        !Trava Produto
        SetDO \Sync, DO_Rc_Fixação_Peça, 0;
        SetDO \Sync, DO_Av_Fixação_Peça, 1;
        !Wait sensores avançado
        WaitTime 1;
        WaitDI DI_Fixa_Peça_1_Rc, 0\MaxTime:= 5\TimeFlag:=timeout_av1;
        WaitDI DI_Fixa_Peça_2_Rc, 0\MaxTime:= 5\TimeFlag:=timeout_av2;
        WaitDI DI_Fixa_Peça_1_Av, 1\MaxTime:= 5\TimeFlag:=timeout_av3;
        WaitDI DI_Fixa_Peça_2_Av, 1\MaxTime:= 5\TimeFlag:=timeout_av4;
        IF (timeout_av1 OR timeout_av2 OR timeout_av3 OR timeout_av4) = TRUE THEN
            PulseDO\PLength:=1, PN_OUT_DO_Cil_NAv;
            TPWrite "Supervisao Sensores, Travas não Avançaram";
            Stop;
            GOTO init_tp;
        ENDIF

    ENDPROC

    !*************************************************************************************************************************
    !Rotinas de Garra: Destravar (Recuar Index Cilindros)
    !*************************************************************************************************************************
    PROC GARRA_DestravarProduto()
    init_dp:
        SetDO PN_OUT_DO_Cil_NRc, 0;

        !Destrava produto na garra
        SetDO \Sync, DO_Av_Fixação_Peça, 0;
        SetDO \Sync, DO_Rc_Fixação_Peça, 1;
        WaitDI DI_Fixa_Peça_1_Av, 0\MaxTime:= 5\TimeFlag:=timeout_rc1;
        WaitDI DI_Fixa_Peça_2_Av, 0\MaxTime:= 5\TimeFlag:=timeout_rc2;
        WaitDI DI_Fixa_Peça_1_Rc, 1\MaxTime:= 5\TimeFlag:=timeout_rc3;
        WaitDI DI_Fixa_Peça_2_Rc, 1\MaxTime:= 5\TimeFlag:=timeout_rc4;
        IF (timeout_rc1 OR timeout_rc2 OR timeout_rc3 OR timeout_rc4) = TRUE THEN
            PulseDO\PLength:=1, PN_OUT_DO_Cil_NRc;
            TPWrite "Supervisao Sensores, Travas não Recuaram";
            Stop;
            GOTO init_dp;
        ENDIF
    ENDPROC

    !*************************************************************************************************************************
    !Rotinas de Garra: Validar Sensor Laser
    !*************************************************************************************************************************
    PROC GARRA_VerificarLaser()
     inicio:
        IF DInput (DI_Pres_Peça_Berço_1) = 0 AND DInput (DI_Pres_Peça_Berço_2) = 1 GOTO Fim;

        PulseDO\PLength:=1, PN_OUT_Produto_Existente;
        TPErase;
        TPWrite "Sensor de presença de peça no berço acionado. Verifique";
        Stop;
        GOTO inicio;

    Fim:
        SetDO PN_OUT_Produto_Existente, 0;
    ENDPROC

    !*************************************************************************************************************************
    !Rotinas de Garra: Validar sensores garra / Garantir que a garra está vazia
    !*************************************************************************************************************************
    PROC GARRA_VerificarGarraVazia()
    !Verifica se robô tem peça na garra ou não

    Verifica:
        IF DI_Pres_Peça_Garra_2 = 1 AND DI_Pres_Peça_Garra_1 = 0 THEN
            GOTO Fim;
        ELSE
            TPErase;
            TPWrite "Deposite manualmente o produto encontrado na garra e reinicie o ciclo";
            TPWrite "Após depositar o produto, adicionar código do produto na IHM";
            IF GInput (PN_IN_Numero_Programa) = 2 THEN
                TPWrite "Programa 'Pega na Esteira de Entrada' necessita de garra vazia para iniciar";
                PulseDO\PLength:=2, PN_OUT_Pos_Home_Manual;
            ELSEIF GInput (PN_IN_Numero_Programa) = 4 THEN
                TPWrite "Programa 'Pega Peça no Buffer' necessita de garra vazia para iniciar";
                PulseDO\PLength:=2, PN_OUT_Pos_Home_Manual;
            ENDIF
            WaitUntil DI_Pres_Peça_Garra_2 = 1 AND DI_Pres_Peça_Garra_1 = 0;
            GOTO Verifica;
        ENDIF
    Fim:
    ENDPROC


    !*************************************************************************************************************************
    !Rotinas de Garra: Define Grip Load da família
    !*************************************************************************************************************************
    PROC GARRA_ConfigurarCarga(Num f)
        TEST f
			CASE 1:
				GripLoad lFamilia_1;
			CASE 2:
				GripLoad lFamilia_2;
			CASE 3:
				GripLoad lFamilia_3;
			CASE 4:
				GripLoad lFamilia_4;

			DEFAULT:
				!Erro
				MsgBoxStop("Número da Família recebida pelo CLP Inexistente!");
				EXIT;
		ENDTEST
    ENDPROC

    !*************************************************************************************************************************
    !Função para ser chamada pela manutenção (retorno para home)
    !*************************************************************************************************************************
    PROC EXTRAS_PosicionaHomeManual()
        VAR robtarget pPosição_Atual;
        VAR num nAux_Limite_Low;

        !Movimente manualmente o robô até uma posição em que esteja livre de colisão e acione os comandos abaixo.

    verif:
        pPosição_Atual := CRobT(\Tool:=tGarra \WObj:=wobj0);

        nAux_Limite_Low := 550;
        IF (pPosição_Atual.trans.z > nAux_Limite_Low) THEN
            GOTO DoHome;
        ELSE
            TPErase;
            TPWrite "Posicione Robô mais Alto";
            Stop\NoRegain;
            GOTO verif;
        ENDIF

    DoHome:
        MoveJ pPosicaoHome, sMov_Geral_Sem_Produto, fine, tGarra \WObj:=wobj0;
        SetDO PN_OUT_Pos_Home_Manual, 0;


    ENDPROC

!*****************************************************************************************************************************
    !FUNÇÕES EXTRAS: Teste de Posições no Buffer (Área "A" - à esquerda do robô quando de costas para as esteiras )
    !*****************************************************************************************************************************
    PROC EXTRAS_TesteBufferAreas()
        !Este programa irá enviar o robô à partir de home, index-por-index (de trás para frente) relacionados às áreas do Buffer


        VAR num f;
        VAR num zLoopValida;
        VAR num zFinal;
        VAR num i_ini;
        VAR num InputUsuarioArea;
        VAR num InputUsuario3Opcoes;

        VAR bool InputUsuarioSim;
        VAR bool InputUsuarioDescer;
        VAR bool init;
        VAR bool SaiLoopValida;
        VAR bool InputUsuarioCrescente;

        VAR robtarget RT_PosicaoBuffer;
        VAR robtarget RT_PosicaoAuxiliar;
        VAR jointtarget RJ_PosicaoAuxiliar;

        VAR speeddata SPEEDDATA_VelocidadeAuxiliar;
        VAR string STR_AreaSelecionada;

        !Considerações iniciais
        TPErase;
        TPWrite "Este programa irá enviar o robô index-por-index. Já deve existir peça na garra!";
        TPWrite "Para sobrescrever os pontos, garanta que foram renomeados de CONST para PERS.";
        Stop;
        TPErase;

        StartMove;

        !Pergunta ao usuário qual família
        f := MsgBoxInputUsuarioModelo();

        !Se usuário cancelou, encerra
        IF f = 5 THEN
            EXIT;
        ENDIF

        !Pergunta ao usuário qual área de trabalho
        !(1=Pallet Entrada, 2=Pallet Saída, 3=A, 4=B, 5=C)
        InputUsuarioArea := MsgBoxInputUsuarioWorkObject();

        TEST InputUsuarioArea
            CASE 3:
                STR_AreaSelecionada := "A";
            CASE 4:
                STR_AreaSelecionada := "B";
            CASE 5:
                STR_AreaSelecionada := "C";
            DEFAULT:
                MsgBoxStop("Função Ainda Não Suportada!");
                EXIT;
        ENDTEST

        !Pergunta ao usuário por qual index começar
        gNUM_IteradorBuffer := MsgBoxInputNumericoUsuario("Qual local do Buffer iniciar? (de 1 a 99). 0 = 'Cancelar'");

        !Se usuário cancelou, encerra
        IF (gNUM_IteradorBuffer = 0) OR (gNUM_IteradorBuffer > 99) THEN
            EXIT;
        ENDIF

        !Pergunta ao usuário se adiciona ou decrementa os indexes
        InputUsuarioCrescente := MsgBoxSimNao("Iterar de forma Crescente ou Decrescente?", "Crescente", "Decrescente");

        !Inicializa Parametros
        AccSet 60, 40;
        MotionSup \On \TuneValue:= 200;

        !Vai pra Home?
        IF MsgBoxSimNao("Retornar para Home?", "Sim", "Não") THEN
            SPEEDDATA_VelocidadeAuxiliar := GetSpeedDataFamilia("SPEEDDATA_Geral", f);
            MoveJ pPosicaoHome, SPEEDDATA_VelocidadeAuxiliar, z500, tGarra\WObj:=wobj0;
        ENDIF

        init := TRUE;

        !index-por-index (de trás para frente)
        WHILE gNUM_IteradorBuffer > 0 DO
            !Verifica se index corresponde à área selecionada (A, B ou C)
            IF GetAreaBuffer(gNUM_IteradorBuffer) <> STR_AreaSelecionada THEN
                GOTO break_a;
            ENDIF

            !Se família HL8, verifica se posição corresponde
            IF (f = 4) AND (NOT IsIndexHL8(gNUM_IteradorBuffer)) THEN
                GOTO break_a;
            ENDIF


            !Lê o valor da posição através da descrição da tag
            RT_PosicaoBuffer := GetPosicaoBuffer(gNUM_IteradorBuffer, f);

            !Lê qual o frame da posição atual
            gWOBJDATA_FrameAtual := GetWObjBuffer(gNUM_IteradorBuffer);


            IF init THEN
                !Vai para centro de massa
                !Ponto intermediario centro de massa
                RT_PosicaoAuxiliar := RT_PosicaoBuffer;
        	    RJ_PosicaoAuxiliar := CalcJointT(RT_PosicaoAuxiliar, tGarra \WObj:=gWOBJDATA_FrameAtual);
                RJ_PosicaoAuxiliar.robax.rax_2 := jposRecolhidoEsteira.robax.rax_2;
                RJ_PosicaoAuxiliar.robax.rax_3 := jposRecolhidoEsteira.robax.rax_3;
                RJ_PosicaoAuxiliar.robax.rax_4 := jposRecolhidoEsteira.robax.rax_4;
                RJ_PosicaoAuxiliar.robax.rax_5 := jposRecolhidoEsteira.robax.rax_5;

                SPEEDDATA_VelocidadeAuxiliar := GetSpeedDataFamilia("SPEEDDATA_Geral", f);
                MoveAbsJ RJ_PosicaoAuxiliar, SPEEDDATA_VelocidadeAuxiliar, z500, tGarra\WObj:=gWOBJDATA_FrameAtual;
                init := false;
            ENDIF


            !Vai para posição acima do local de deposita
            RT_PosicaoAuxiliar := RT_PosicaoBuffer;
            RT_PosicaoAuxiliar.trans.z := RT_PosicaoAuxiliar.trans.z + 450;

            SPEEDDATA_VelocidadeAuxiliar := GetSpeedDataFamilia("SPEEDDATA_Geral", f);
            MoveL RT_PosicaoAuxiliar, SPEEDDATA_VelocidadeAuxiliar, z20, tGarra\WObj:=gWOBJDATA_FrameAtual;

            !Ponto acima do berço (seguro)
            RT_PosicaoAuxiliar := RT_PosicaoBuffer;
            RT_PosicaoAuxiliar.trans.z := RT_PosicaoAuxiliar.trans.z + 300;

            SPEEDDATA_VelocidadeAuxiliar := GetSpeedDataFamilia("SPEEDDATA_Geral", f);
            MoveL RT_PosicaoAuxiliar, SPEEDDATA_VelocidadeAuxiliar, z50, tGarra\WObj:=gWOBJDATA_FrameAtual;

            !Aqui já temos uma boa idéia se irá entrar sem bater.
            !Se precisar de algum ajuste, usuário poderá fazê-lo e confirmar
            StopMove;

            ClearPath;
            !InputUsuarioSim := MsgBoxSimNao("Ajustar a posição de entrada e confirmar para prosseguir", "Prosseguir", "Cancelar");
            MsgBoxStop("Ajustar a posição de entrada. Aperte 'Play' para prosseguir");
            StartMove;

            !Ponto de aproximação
            AccSet 30, 40;
            MotionSup \On \TuneValue:= 80;

            !Parte-se do princípio que usuário alterou a posição relativa
            !Pega posição atual e altera Z para bater com a posição do buffer
            RT_PosicaoAuxiliar := CRobT(\Tool:=tGarra \WObj:=gWOBJDATA_FrameAtual);
            RT_PosicaoAuxiliar.trans.z := RT_PosicaoBuffer.trans.z + 55;

            SPEEDDATA_VelocidadeAuxiliar := GetSpeedDataFamilia("SPEEDDATA_AtaqueLinSeg", f);
            MoveL RT_PosicaoAuxiliar, SPEEDDATA_VelocidadeAuxiliar, z0, tGarra\WObj:=gWOBJDATA_FrameAtual;

            !Registra Z original do ponto em questão
            zFinal := RT_PosicaoBuffer.trans.z;

            !Aqui já temos uma boa idéia se irá entrar sem bater.
            !Se precisar de algum ajuste, usuário poderá fazê-lo e confirmar

            StopMove;
            ClearPath;
            InputUsuario3Opcoes := MsgBox3Opcoes("Ajustar posição. Selecionar Opção:", "Descer 5mm", "Pular", "Descer Posição Final");
            StartMove;

            If InputUsuario3Opcoes <> 2 THEN
                SaiLoopValida := FALSE;
            ELSE
                SaiLoopValida := TRUE;
            ENDIF

            !Agora entra em loop, decrementando Z e perguntando input do usuário
            WHILE NOT SaiLoopValida DO

                !Parte-se do princípio que usuário alterou a posição relativa
                !Pega posição atual e altera Z para bater com a posição do buffer
                RT_PosicaoAuxiliar := CRobT(\Tool:=tGarra \WObj:=gWOBJDATA_FrameAtual);

                TEST InputUsuario3Opcoes
                    CASE 1: !Desce 5mm
                        RT_PosicaoAuxiliar.trans.z := RT_PosicaoAuxiliar.trans.z - 5;
                    CASE 3: !Desce ao final
                        RT_PosicaoAuxiliar.trans.z := zFinal;
                    DEFAULT: !Erro
                        MsgBoxStop("Algo deu errado.");
                ENDTEST

                SPEEDDATA_VelocidadeAuxiliar := GetSpeedDataFamilia("SPEEDDATA_AtaqueLinCol", f);
                MoveL RT_PosicaoAuxiliar, SPEEDDATA_VelocidadeAuxiliar, fine, tGarra\WObj:=gWOBJDATA_FrameAtual;

                zLoopValida := RT_PosicaoAuxiliar.trans.z - 5;
                !Segue somente se ainda podemos descer
                IF zLoopValida >= zFinal THEN
                    !Novamente pergunta ao usuário se pode continuar
                    !Se precisar de algum ajuste, usuário poderá fazê-lo e confirmar

                    StopMove;
                    ClearPath;
                    InputUsuario3Opcoes := MsgBox3Opcoes("Ajustar posição. Selecionar Opção:", "Descer 5mm", "Pular", "Descer Posição Final");
                    StartMove;

                    !Se usuário pediu para registrar, encerra
                    IF InputUsuario3Opcoes = 2 THEN
                        SaiLoopValida := TRUE;
                    ENDIF
                ELSE
                    SaiLoopValida := TRUE;
                ENDIF

            ENDWHILE


            StopMove;
            ClearPath;
            InputUsuario3Opcoes := MsgBox3Opcoes("Robô na posição " + NumToStr(gNUM_IteradorBuffer, 0) + "(Família " + NumToStr(f, 0) + "). Registrar Nova Posição?", "Registrar", "Prosseguir Sem Registrar", "Testar Garra Abre/Fecha");
            StartMove;

            !Aqui usuário alterou a posição do robô e pediu para sobrescrevê-la
            TEST InputUsuario3Opcoes
                    CASE 1: !Registrar
                        SetPosicaoBuffer gNUM_IteradorBuffer, f, CRobT(\Tool:=tGarra \WObj:=gWOBJDATA_FrameAtual);
                    CASE 2:
                        !Pula
                    CASE 3: !Teste de Garra
                        !Fazer!
                    DEFAULT: !Erro
                        MsgBoxStop("Algo deu errado.");
                ENDTEST

            !Usuário deu sequência: Sobe Garra Lentamente
            RT_PosicaoAuxiliar := CRobT(\Tool:=tGarra \WObj:=gWOBJDATA_FrameAtual);
            RT_PosicaoAuxiliar.trans.z := RT_PosicaoAuxiliar.trans.z + 50;

            SPEEDDATA_VelocidadeAuxiliar := GetSpeedDataFamilia("SPEEDDATA_RecuoLinCol", f);
            MoveL RT_PosicaoAuxiliar, SPEEDDATA_VelocidadeAuxiliar, z5, tGarra\WObj:=gWOBJDATA_FrameAtual;

            !Usuário deu sequência: Sobe Garra Mais rápido e segue p/ próximo ponto
            RT_PosicaoAuxiliar.trans.z := RT_PosicaoAuxiliar.trans.z + 350;

            SPEEDDATA_VelocidadeAuxiliar := GetSpeedDataFamilia("SPEEDDATA_RecuoLinSeg", f);
            MoveL RT_PosicaoAuxiliar, SPEEDDATA_VelocidadeAuxiliar, z5, tGarra\WObj:=gWOBJDATA_FrameAtual;

            break_a:

            !Inc/Dec iterador
            IF InputUsuarioCrescente THEN
                gNUM_IteradorBuffer := gNUM_IteradorBuffer +1;
            ELSE
                gNUM_IteradorBuffer := gNUM_IteradorBuffer -1;
            ENDIF
        ENDWHILE

    ENDPROC

    !*****************************************************************************************************************************
    !Retorna um texto contendo o nome do tipo para mensagens no TP
    !*****************************************************************************************************************************
    FUNC string GetModelo(Num i)
        TEST i
            CASE 1:
                RETURN "HL2 (1)";
            CASE 2:
                RETURN "HL4 (2)";
            CASE 3:
                RETURN "HL6 (3)";
            CASE 4:
                RETURN "HL8 (4)";
            DEFAULT :
                RETURN "?";
        ENDTEST
    ENDFUNC

    !*****************************************************************************************************************************
    !Lança Mensagem na Tela e Aguarda Usuário Selecionar o Modelo (de 1 a 4). Retorno = 5 significa usuário cancelou a rotina
    !*****************************************************************************************************************************
    FUNC num MsgBoxInputUsuarioModelo()
        VAR num NUM_RespostaTP;

        TPErase;
        TPReadFK NUM_RespostaTP, "Indicar Qual o Modelo:", "HL2 (1)", "HL4 (2)", "HL6 (3)", "HL8 (4)", "Cancelar!";
        RETURN NUM_RespostaTP;

    ENDFUNC

    !*****************************************************************************************************************************
    !Lança Mensagem na Tela e Aguarda Usuário Selecionar o Work Object(de 1 a 5)
    !1=Pallet Entrada, 2=Pallet Saída, 3=A, 4=B, 5=C
    !*****************************************************************************************************************************
    FUNC num MsgBoxInputUsuarioWorkObject()
        VAR num NUM_RespostaTP;

        TPErase;
        TPReadFK NUM_RespostaTP, "Indicar Qual a Área de Trabalho (Work Object):", "Pallet Entrada", "Pallet Saída", "Buffer A", "Buffer B", "Buffer C";
        RETURN NUM_RespostaTP;

    ENDFUNC

    !*****************************************************************************************************************************
    !Lança Mensagem na Tela (configurável) e Aguarda Usuário entrar um valor qualquer
    !*****************************************************************************************************************************
    FUNC num MsgBoxInputNumericoUsuario(string pSTR_Msg)
        VAR num NUM_RespostaTP;

        TPErase;
        TPReadNum  NUM_RespostaTP, pSTR_Msg;
        RETURN NUM_RespostaTP;

    ENDFUNC

    !*****************************************************************************************************************************
    !Lança Mensagem na Tela e Para Execução do Programa (Usuário poderá retornar execução normalmente com um "play"
    !*****************************************************************************************************************************
    PROC MsgBoxStop(string pSTR_msg)
        VAR NUM lNUM_RespostaUsuario;

        TPErase;
        TPWrite pSTR_msg;
        Stop;
        TPErase;

    ENDPROC

    !*****************************************************************************************************************************
    !Lança Mensagem na Tela e Aguarda Usuário apertar "Ok"
    !*****************************************************************************************************************************
    PROC MsgBoxOk(string pSTR_msg)
        VAR NUM lNUM_RespostaUsuario;

        TPErase;
        TPReadFK lNUM_RespostaUsuario, pSTR_msg, stEmpty, stEmpty, stEmpty, stEmpty, "Ok";
    ENDPROC

    !*****************************************************************************************************************************
    !Lança Mensagem na Tela e Retorna "true" se usuário apertou "sim"
    !*****************************************************************************************************************************
    FUNC bool MsgBoxSimNao(string pSTR_Msg, string pSTR_Sim, string pSTR_Nao)
        VAR NUM lNUM_RespostaUsuario;

        TPErase;
        TPReadFK lNUM_RespostaUsuario, pSTR_Msg, pSTR_Nao, stEmpty, stEmpty, stEmpty, pSTR_Sim;

        IF lNUM_RespostaUsuario = 5 THEN
            RETURN TRUE;
        ELSE
            RETURN FALSE;
        ENDIF

    ENDFUNC

    !*****************************************************************************************************************************
    !Lança Mensagem na Tela Com 3 Opções. Retorna 1,2,3
    !*****************************************************************************************************************************
    FUNC Num MsgBox3Opcoes(string pSTR_Msg, string pSTR_Opcao1, string pSTR_Opcao2, string pSTR_Opcao3)
        VAR num lNUM_RespostaUsuario;

        TPErase;
        TPReadFK lNUM_RespostaUsuario, pSTR_Msg, pSTR_Opcao1, pSTR_Opcao2, pSTR_Opcao3, stEmpty, stEmpty;
        TPErase;

        RETURN lNUM_RespostaUsuario;

    ENDFUNC

    !*************************************************************************************************************************
    !*************************************************************************************************************************
    !*************************************************************************************************************************
    !FUNÇÕES NÃO MAIS UTILIZADAS
    PROC Z_OLD_VerificacaoInicial ()
        VAR num Passo_Verif_Inic;
        VAR num RespostaTP;
        CONST pos pOffset_Esteiras_Z := [0,0,300];
        CONST pos pOffset_Esteiras_XZ := [100,0,300];

        VAR robtarget pPosição_Atual;
    inicio:

        !Verifica posição atual do robô
        pPosição_Atual := CRobT(\Tool:=tGarra \WObj:=wobj0);

        IF pPosição_Atual.extax.eax_a > 2700 AND pPosição_Atual.trans.x < -1700 THEN
            Passo_Verif_Inic := 10;
            GOTO Analise;
        ENDIF

        IF pPosição_Atual.trans.x < 650 THEN
            Passo_Verif_Inic := 20;
        ENDIF

        IF pPosição_Atual = pPosicaoHome THEN
            GOTO Final;
        ENDIF

        Passo_Verif_Inic := 30;

   Analise:

        !****************************************************************!
        !               ANALISA O QUE FAZER EM CADA CASO                 !
        !****************************************************************!
        ! Passo_Verif_Inic = 10 - Acima das Esteiras                     !
        ! Passo_Verif_Inic = 20 - Abaixo região segura acima dos berços  !
        ! Passo_Verif_Inic = 30 - Demais regiões                         !
        !****************************************************************!

        TEST Passo_Verif_Inic

        CASE 10:
            !Verifica presença de peça na garra
            IF (DI_Pres_Peça_Garra_2 = 1 AND DI_Pres_Peça_Garra_1 = 0) OR (DI_Pres_Peça_Garra_1 = 1 OR DI_Pres_Peça_Garra_2 = 0 AND DI_Fixa_Peça_1_Rc = 1 AND DI_Fixa_Peça_2_Rc = 1 AND PN_IN_Garra_Aberta = 1) OR (DI_Pres_Peça_Garra_1 = 1 OR DI_Pres_Peça_Garra_2 = 0 AND DI_Fixa_Peça_1_Av = 1 AND DI_Fixa_Peça_2_Av = 1 AND PN_IN_Garra_Fechada = 1) THEN
                GOTO movimento_esteiras;
            ENDIF

            IF DI_Pres_Peça_Garra_1 = 1 OR DI_Pres_Peça_Garra_2 = 0 AND ((DI_Fixa_Peça_1_Rc = 1 OR DI_Fixa_Peça_2_Rc = 1) AND (PN_IN_Garra_Fechada = 1 OR PN_IN_Garra_Aberta = 0)) THEN
                TPReadFK RespostaTP, "Garanta manualmente garra em condições de movimentação e pressione OK", stEmpty, stEmpty, stEmpty, stEmpty, "OK";
                IF (RespostaTP = 5 OR RespostaTP = 0) GOTO inicio;
            ENDIF

    movimento_esteiras:

            pPosição_Desejada := pPosição_Atual;
            pPosição_Desejada.trans := pPosição_Desejada.trans + pOffset_Esteiras_Z;
            MoveL pPosição_Desejada, v30, z10, tGarra \WObj:=wobj0;

            pPosição_Desejada := pPosição_Atual;
            pPosição_Desejada.trans := pPosição_Desejada.trans + pOffset_Esteiras_XZ;
            MoveL pPosição_Desejada, v30, z10, tGarra \WObj:=wobj0;

            GOTO Final;

        CASE 20:
            !Verifica presença de peça na garra
            IF (DI_Pres_Peça_Garra_2 = 1 AND DI_Pres_Peça_Garra_1 = 0) OR (DI_Pres_Peça_Garra_1 = 1 OR DI_Pres_Peça_Garra_2 = 0 AND DI_Fixa_Peça_1_Rc = 1 AND DI_Fixa_Peça_2_Rc = 1 AND PN_IN_Garra_Aberta = 1) OR (DI_Pres_Peça_Garra_1 = 1 OR DI_Pres_Peça_Garra_2 = 0 AND DI_Fixa_Peça_1_Av = 1 AND DI_Fixa_Peça_2_Av = 1 AND PN_IN_Garra_Fechada = 1) THEN
                GOTO movimento_berços;
            ENDIF

            IF DI_Pres_Peça_Garra_1 = 1 OR DI_Pres_Peça_Garra_2 = 0 AND ((DI_Fixa_Peça_1_Rc = 1 OR DI_Fixa_Peça_2_Rc = 1) AND (PN_IN_Garra_Fechada = 1 OR PN_IN_Garra_Aberta = 0))  THEN !Falta sinal garra aberta
                TPReadFK RespostaTP, "Garanta manualmente garra em condições de movimentação e pressione OK", stEmpty, stEmpty, stEmpty, stEmpty, "OK";
                IF (RespostaTP = 5 OR RespostaTP = 0) GOTO inicio;
            ENDIF

        movimento_berços:

            pPosição_Desejada := pPosição_Atual;
            pPosição_Desejada.trans.z := 660;
            MoveL pPosição_Desejada, v30, z10, tGarra \WObj:=wobj0;

            GOTO Final;

        CASE 30:

            !Verifica presença de peça na garra
            IF (DI_Pres_Peça_Garra_2 = 1 AND DI_Pres_Peça_Garra_1 = 0) OR (DI_Pres_Peça_Garra_1 = 1 OR DI_Pres_Peça_Garra_2 = 0 AND DI_Fixa_Peça_1_Rc = 1 AND DI_Fixa_Peça_2_Rc = 1 AND PN_IN_Garra_Aberta = 1) OR (DI_Pres_Peça_Garra_1 = 1 OR DI_Pres_Peça_Garra_2 = 0 AND DI_Fixa_Peça_1_Av = 1 AND DI_Fixa_Peça_2_Av = 1 AND PN_IN_Garra_Fechada = 1) THEN
                GOTO Final;
            ENDIF

            IF DI_Pres_Peça_Garra_1 = 1 OR DI_Pres_Peça_Garra_2 = 0 AND ((DI_Fixa_Peça_1_Rc = 1 OR DI_Fixa_Peça_2_Rc = 1) AND (PN_IN_Garra_Fechada = 1 OR PN_IN_Garra_Aberta = 0))  THEN !Falta sinal garra aberta
                TPReadFK RespostaTP, "Garanta manualmente garra em condições de movimentação e pressione OK", stEmpty, stEmpty, stEmpty, stEmpty, "OK";
                IF (RespostaTP = 5 OR RespostaTP = 0) GOTO inicio;
            ENDIF

        DEFAULT:

            TPErase;
            TPWrite "Não foi possível localizar o robô. Movimente manualmente para a posição inicial";
            Stop;
            GOTO inicio;

        ENDTEST

   Final:
        Passo_Verif_Inic := 0;

        !Se em posição inicial e não foi solicitada parada, encerra rotina
        IF pPosição_Atual = pPosicaoHome GOTO Fim;

        !Vai para posição de trabalho
        MoveJ pPosicaoHome, sMov_Geral_Com_Produto, fine, tGarra \WObj:=wobj0;

   Fim:
    ENDPROC


    !*************************************************************************************************************************
    !FUNÇÕES EXTRAS: Movimenta Para o Angulo Zero de cada eixo
    !*************************************************************************************************************************
    PROC EXTRAS_MovimentaEixosZero()
      !Ponto Zero do Robo...
      MoveAbsJ [[0,0,0,0,0,0],[0,9E+09,9E+09,9E+09,9E+09,9E+09]] \NoEOffs, v400, fine, tool0;
      !
	ENDPROC

    !*************************************************************************************************************************
    !FUNÇÕES EXTRAS: Teste do 7o eixo
    !*************************************************************************************************************************
    PROC EXTRAS_Teste7oEixo()
        CONST robtarget pPos1:=[[1782.23,-9.35,841.69],[0.0118043,0.0684442,-0.99757,-0.00543028],[-1,0,-1,0],[2708.4,9E+09,9E+09,9E+09,9E+09,9E+09]];
        CONST robtarget pPos2:=[[1782.23,-9.35,841.69],[0.0118043,0.0684442,-0.99757,-0.00543028],[-1,0,-1,0],[-2708.4,9E+09,9E+09,9E+09,9E+09,9E+09]];

        WHILE TRUE DO
            MoveL pPos1, v5000, z50, tGarra\WObj:=wobj0;
            MoveL pPos2, v5000, z50, tGarra\WObj:=wobj0;
        ENDWHILE

    ENDPROC





    !*************************************************************************************************************************
    !*************************************************************************************************************************
    !*************************************************************************************************************************
    !FUNÇÕES NÃO MAIS UTILIZADAS


	PROC Z_OLD_TesteEixo1()
		MoveJ [[4357.31,-1398.45,1978.14],[0.687563,0.27921,0.236299,0.627265],[-1,0,1,1],[2346.44,9E+09,9E+09,9E+09,9E+09,9E+09]], v2500, z50, tGarra\WObj:=FRAME_BufferA;
		WaitTime\InPos, 1;
		MoveJ [[3711.49,-1299.99,468.29],[0.0309804,-0.747554,-0.66329,0.0158269],[-1,0,1,0],[2346.44,9E+09,9E+09,9E+09,9E+09,9E+09]], v2500, z50, tGarra\WObj:=FRAME_BufferA;
		WaitTime\InPos, 1;
	ENDPROC

    PROC Z_OLD_Routine1()
		pMov_Pega_Depos_Buffer := pPega_Esteira_Entrada_Fam_1;
        pMov_Pega_Depos_Buffer.trans := pMov_Pega_Depos_Buffer.trans + [0,0,500];
        MoveJ pMov_Pega_Depos_Buffer, v1000, fine, tGarra\WObj:=FRAME_BufferA;
        MoveL pPega_Esteira_Entrada_Fam_1, v200, fine, tGarra\WObj:=FRAME_BufferA;
        MoveL pMov_Pega_Depos_Buffer, v2500, fine, tGarra\WObj:=FRAME_BufferA;
        MoveJ pPosicaoHome, v1000, fine, tGarra\WObj:=wobj0;
	ENDPROC

    PROC Z_OLD_TesteAfericao()
      !Ponto de Referencia p/ troca de lagarto..
      MoveJ pCheck_00,v500,z30,tGarra\WObj:=wobj0;
      MoveJ pCheck_01,v500,z30,tGarra\WObj:=wobj0;
      MoveJ pCheck_02,v500,z30,tGarra\WObj:=wobj0;
      MoveL Offs(pCheck,0,0,400),v500,z30,tGarra\WObj:=wobj0;
      MoveL Offs(pCheck,0,0,100), v200, z30, tGarra\WObj:=wobj0;
      MoveL Offs(pCheck,0,0,40), v40, z5, tGarra\WObj:=wobj0;
      MoveL pCheck, v20, fine, tGarra\WObj:=wobj0;
      WaitUntil\InPos,TRUE;
      WaitTime\InPos, 1.5;
      !Stop;
      MoveL Offs(pCheck,0,0,40),v100,z5,tGarra\WObj:=wobj0;
      MoveL Offs(pCheck,0,0,100),v400,z30,tGarra\WObj:=wobj0;
      MoveL Offs(pCheck,0,0,400),v500,z30,tGarra\WObj:=wobj0;
      MoveJ pCheck_02,v500,z30,tGarra\WObj:=wobj0;
      MoveJ pCheck_01,v500,z30,tGarra\WObj:=wobj0;
      MoveJ pCheck_00,v500,z30,tGarra\WObj:=wobj0;
      !
    ENDPROC

ENDMODULE
